TYPE "MEStoPLC_SubCheckIn_ext"
VERSION : 0.1
   STRUCT
      Spare : Byte;
      Load_SubPart1OK : Bool;
      Load_SubPart1tNG : Bool;
      Load_SubPart1ReqMesDone : Bool;
      SubPart1Spare : Bool;
      SubPart1Spare1 : Bool;
      SubPart1Spare2 : Bool;
      SubPart1Spare3 : Bool;
      SubPart1Spare4 : Bool;
      Load_SubPart2OK : Bool;
      Load_SubPart2tNG : Bool;
      Load_SubPart2ReqMesDone : Bool;
      SubPart2Spare : Bool;
      SubPart2Spare1 : Bool;
      SubPart2Spare2 : Bool;
      SubPart2Spare3 : Bool;
      SubPart2Spare4 : Bool;
      Load_SubPart3OK : Bool;
      Load_SubPart3tNG : Bool;
      Load_SubPart3ReqMesDone : Bool;
      SubPart3Spare : Bool;
      SubPart3Spare1 : Bool;
      SubPart3Spare2 : Bool;
      SubPart3Spare3 : Bool;
      SubPart3Spare4 : Bool;
      Load_SubPart4OK : Bool;
      Load_SubPart4tNG : Bool;
      Load_SubPart4ReqMesDone : Bool;
      SubPart4Spare : Bool;
      SubPart4Spare1 : Bool;
      SubPart4Spare2 : Bool;
      SubPart4Spare3 : Bool;
      SubPart4Spare4 : Bool;
      Load_SubPart5OK : Bool;
      Load_SubPart5tNG : Bool;
      Load_SubPart5ReqMesDone : Bool;
      SubPart5Spare : Bool;
      SubPart5Spare1 : Bool;
      SubPart5Spare2 : Bool;
      SubPart5Spare3 : Bool;
      SubPart5Spare4 : Bool;
      Load_SubPart6OK : Bool;
      Load_SubPart6tNG : Bool;
      Load_SubPart6ReqMesDone : Bool;
      SubPart6Spare : Bool;
      SubPart6Spare1 : Bool;
      SubPart6Spare2 : Bool;
      SubPart6Spare3 : Bool;
      SubPart6Spare4 : Bool;
      Load_SubPart7OK : Bool;
      Load_SubPart7tNG : Bool;
      Load_SubPart7ReqMesDone : Bool;
      SubPart7Spare : Bool;
      SubPart7Spare1 : Bool;
      SubPart7Spare2 : Bool;
      SubPart7Spare3 : Bool;
      SubPart7Spare4 : Bool;
      Load_SubPart8OK : Bool;
      Load_SubPart8tNG : Bool;
      Load_SubPart8ReqMesDone : Bool;
      SubPart8Spare : Bool;
      SubPart8Spare1 : Bool;
      SubPart8Spare2 : Bool;
      SubPart8Spare3 : Bool;
      SubPart8Spare4 : Bool;
      SpareByte : Byte;
   END_STRUCT;

END_TYPE

